TYPE ST_EasyTempPara :
STRUCT
	bTuned : BOOL;
	stPID : ST_CTRL_ParaController;
	stPara: ST_CTRL_TempCtrlParameter;
END_STRUCT
END_TYPE

(* stored: Version 1.1.0.1, ProductVersion 3.1.4024.12
   DUT ST_EasyTempPara: Id {edc06a74-c9cb-47a6-89cb-bcc758dcb537} *)
